TYPE tstCTCConfigVariable :
STRUCT
	Name 			:STRING[64];
	Index 			:WORD;
	Subindex 		:BYTE;
	DataType 		:USINT := 0; 	// 0=Real, 1=Usint
	ValueIfReal 	:REAL;
	ValueIfUSINT 	:USINT;
END_STRUCT
END_TYPE

(* stored: Version 1.1.0.1, ProductVersion 3.1.4026.17
   DUT tstCTCConfigVariable: Id {3149f17d-b353-4617-955f-2524210527ec} *)
